// TwinCAT 3 PLC project TcLog
// Title: TcLog
// Company: Benedikt Geisler
// Author: Benedikt Geisler
// ProjectVersion: 0.2.2
// Description: TcLog provides logging functionality to TwinCAT.
// ProgramVersion: 3.1.4023.0
// libraries:
//   Base Interfaces,newest,System
//   Tc2_Standard, * (Beckhoff Automation GmbH)
//   Tc2_System, * (Beckhoff Automation GmbH)
//   Tc2_Utilities, * (Beckhoff Automation GmbH)
//   Tc3_DynamicMemory, * (Beckhoff Automation GmbH)
//   Tc3_Module, * (Beckhoff Automation GmbH)
// project tree:
//   / CONSTANTS.TcGVL
//   Helper functions/ ANY_TO_STRING2.TcPOU, DeleteOldFiles.TcPOU, DynamicStringBuffer.TcPOU, GenerateTimeData.TcPOU, GetFileAgeInSeconds.TcPOU
//   Helper functions/_DataTypes/ DeleteFilesState.TcDUT, PersistToFileState.TcDUT (not stored)
//   Logger/DUT/ E_ErrorCode.TcDUT, E_LogLevel.TcDUT, E_RollingInterval.TcDUT, ST_Error.TcDUT, ST_LoggingConfiguration.TcDUT
//   Logger/ITF/ ILog.TcIO, ILogCore.TcIO
//   Logger/POU/ LogLevel_To_AdsLogMsgType.TcPOU, TcLog.TcPOU, TcLogCore.TcPOU, TcLogTRIG.TcPOU
//   StringBuilder/ ILimitedStringBuilder.TcIO, IStringBuilder.TcIO, StringBuilder.TcPOU
//   Version/ Global_Version.TcGVL
// (motion and I/O tree: see PLC project tclogtest)
// real-time tasks:
//   TASK PlcTask: cycle T#10ms, priority 20, ADS port 350

// ---- Helper functions/_DataTypes/DeleteFilesState.TcDUT
{attribute 'qualified_only'}
{attribute 'strict'}
TYPE INTERNAL DeleteFilesState :
(
	Idle := 0,
  SearchNextFile,
  WaitUntilExecutionDone,
  ProcessFoundFiles,
  CheckIfFileIsDirectory,
  CheckFileTime,
  DeleteFile,
  FileDeleted
);
END_TYPE

// ---- Logger/DUT/E_ErrorCode.TcDUT
{attribute 'qualified_only'}
{attribute 'strict'}
{attribute 'to_string'}
// Provides error return codes for TcLogCore
TYPE E_ErrorCode : 
(
	None,
	OpeningFileFailed,
	WritingToFileFailed,
	ClosingFileFailed,
	EnumeratingFilesInSpecifiedDirectoryFailed,
	DeletingFileFailed,
	FifoOverflow
);
END_TYPE

// ---- Logger/DUT/E_LogLevel.TcDUT
{attribute 'qualified_only'}
{attribute 'strict'}
{attribute 'to_string'}
// Log level of message to be logged.
TYPE E_LogLevel :
(
	Debug,
	Information,
	Warning,
	Error,
	Fatal
);
END_TYPE

// ---- Logger/DUT/E_RollingInterval.TcDUT
{attribute 'qualified_only'}
{attribute 'strict'}
{attrivute 'to_string'}
// Rolling interval to create a new log file when expired. 
TYPE E_RollingInterval :
(
	None,
	Hourly,
	Daily,
	Monthly
);
END_TYPE

// ---- Logger/DUT/ST_Error.TcDUT
TYPE ST_Error :
STRUCT
	Active : BOOL; // TRUE = error is active
	Code : INT; // Error return code => E_ErrorCode
	Info : Tc2_System.T_MaxString; // Error message
END_STRUCT
END_TYPE

// ---- Logger/DUT/ST_LoggingConfiguration.TcDUT
// Configuration of TcLog
TYPE ST_LoggingConfiguration :
STRUCT
	FileName : STRING;
	FilePath : Tc2_System.T_MaxString;
	IncludeInstancePath : BOOL;
	WriteToAds : BOOL;
	RollingInterval : E_RollingInterval;
	MinimumLevel : E_LogLevel;
	Delimiter : STRING(1);
	LogFileLifespan : UINT;
	TimestampFormat : STRING;
END_STRUCT
END_TYPE

// ---- CONSTANTS.TcGVL
{attribute 'qualified_only'}
VAR_GLOBAL CONSTANT
	BUFFER_SIZE : INT := (100 * UDINT_TO_INT(MAX_STRING_LENGTH));
END_VAR

// ---- Version/Global_Version.TcGVL
{attribute 'TcGenerated'}
{attribute 'no-analysis'}
{attribute 'linkalways'}
// This function has been automatically generated from the project information.
VAR_GLOBAL CONSTANT
	{attribute 'const_non_replaced'}
	stLibVersion_TcLog : ST_LibVersion := (iMajor := 0, iMinor := 2, iBuild := 2, iRevision := 0, nFlags := 1, sVersion := '0.2.2');
END_VAR

// ---- Logger/ITF/ILog.TcIO
INTERFACE ILog

METHOD SetLogger : BOOL
VAR_INPUT
	Ref2Core : ILogCore;
END_VAR
END_METHOD

END_INTERFACE

// ---- Logger/ITF/ILogCore.TcIO
INTERFACE ILogCore

// Logger method.
// Logs data in custom format. No additional formatting will be done.
METHOD LogCustomFormat : BOOL
VAR_INPUT
	Data : Tc2_System.T_MaxString; // Data to be logged. No additional formatting will be done.
END_VAR
END_METHOD

// Logger method.
// Logs in the standard format. This includes
// - timestamp
// - log level
// - log message
// - instance path of logging source (optional)
// The message will only be logged if the logging level exceeds the configured minimum logging level.
METHOD LogStandardFormat : BOOL
VAR_INPUT
	Data : Tc2_System.T_MaxString; // Data to be logged. Additional formatting wil be done.
	InstancePath : Tc2_System.T_MaxString; // Instance path of calling logger to locate source of logging message.
	LogLevel : E_LogLevel; // Log level of message.
END_VAR
END_METHOD

END_INTERFACE

// ---- StringBuilder/ILimitedStringBuilder.TcIO
INTERFACE INTERNAL ILimitedStringBuilder

METHOD Append : IStringBuilder // Append text TO t current build STRING.
VAR_INPUT
    Text : Tc2_System.T_MaxString; //Text to append to current build string
END_VAR
END_METHOD

METHOD AppendIf : IStringBuilder
VAR_INPUT
    Condition : BOOL;
    Text : Tc2_System.T_MaxString;
END_VAR
END_METHOD

METHOD Reset : ILimitedStringBuilder //Reset current build STRING TO an empty STRING.
END_METHOD

METHOD ToString : Tc2_System.T_MaxString //Returns current build STRING.
END_METHOD

END_INTERFACE

// ---- StringBuilder/IStringBuilder.TcIO
INTERFACE IStringBuilder

METHOD  Append : IStringBuilder // Append text to t current build string.
VAR_INPUT
	text : Tc2_System.T_MaxString; //Text to append to current build string
END_VAR
END_METHOD

METHOD AppendIf : IStringBuilder
VAR_INPUT
	condition	:	BOOL;
	text : Tc2_System.T_MaxString;
END_VAR
END_METHOD

METHOD InsertAtLocation : IStringBuilder
VAR_INPUT
	Text : Tc2_System.T_MaxString;
	Position:INT;
END_VAR
END_METHOD

METHOD PadLeft : IStringBuilder
VAR_INPUT
	text : Tc2_System.T_MaxString; // Text to append to current build string
	length : INT; // Total length of text + padding
	char : STRING(1); // Character to be padded left of text
END_VAR
END_METHOD

METHOD Reset : ILimitedStringBuilder //Reset current build string to an empty string.
END_METHOD

METHOD ToString : Tc2_System.T_MaxString //Returns current build string.
END_METHOD

END_INTERFACE

// ---- Helper functions/ANY_TO_STRING2.TcPOU
// Converts value of ANY to String.
FUNCTION ANY_TO_STRING2 : T_MAXSTRING
VAR_INPUT
	Data:	ANY;
END_VAR
VAR
	pAnyReal : POINTER TO REAL;
	pAnyLReal: POINTER TO LREAL;	
	pAnyDateAndTime : POINTER TO DATE_AND_TIME;
	pAnyDate: POINTER TO DATE;
	pAnyTime: POINTER TO TIME;
	pAnyWString: POINTER TO WSTRING;
	pAnyTOD: POINTER TO TOD;
	pAnyString: POINTER TO STRING;
	sString: T_MAXSTRING;
	wWString: WSTRING;
END_VAR

IF Data.TypeClass = __SYSTEM.TYPE_CLASS.TYPE_REAL THEN
	pAnyReal := Data.pValue;
	ANY_TO_STRING2 := REAL_TO_STRING(pAnyReal^);
	
ELSIF Data.TypeClass = __SYSTEM.TYPE_CLASS.TYPE_LREAL THEN
	pAnyLReal := Data.pValue;
	ANY_TO_STRING2 := LREAL_TO_STRING(pAnyLReal^);
	
ELSIF Data.TypeClass = __SYSTEM.TYPE_CLASS.TYPE_DATEANDTIME THEN
	pAnyDateAndTime := Data.pValue;
	ANY_TO_STRING2 := DT_TO_STRING(pAnyDateAndTime^);	
	
ELSIF Data.TypeClass = __SYSTEM.TYPE_CLASS.TYPE_DATE THEN
	pAnyDate := Data.pValue;
	ANY_TO_STRING2 := DATE_TO_STRING(pAnyDate^);
	
ELSIF Data.TypeClass = __SYSTEM.TYPE_CLASS.TYPE_TIME THEN
	pAnyTime := Data.pValue;
	ANY_TO_STRING2 := TIME_TO_STRING(pAnyTime^);
	
ELSIF Data.TypeClass = __SYSTEM.TYPE_CLASS.TYPE_STRING THEN
	pAnyString := Data.pValue;
	ANY_TO_STRING2 := pAnyString^;
	
ELSIF Data.TypeClass = __SYSTEM.TYPE_CLASS.TYPE_WSTRING THEN
	pAnyWString := Data.pValue;
	wWString := pAnyWString^;
	WSTRING_TO_STRING2(ADR(sString), ADR(wWstring), SIZEOF(wWString));
	ANY_TO_STRING2 := sString;
	
ELSIF Data.TypeClass = __SYSTEM.TYPE_CLASS.TYPE_TIMEOFDAY THEN
	pAnyTOD := Data.pValue;
	ANY_TO_STRING2 := TOD_TO_STRING(pAnyTOD^);
	
ELSE
	ANY_TO_STRING2 := ANY_TO_STRING(Data.pValue^);
END_IF

END_FUNCTION

// ---- Helper functions/DeleteOldFiles.TcPOU
FUNCTION_BLOCK DeleteOldFiles
VAR_INPUT
	StartScan : BOOL; // Rising edge starts scan for out-of-date log files and deletes them.
	ExpirationInDays : UINT; // Files will be deleted if older than n days
	FilePath : Tc2_System.T_MaxString; // Path to files to be deleted
	FileName : Tc2_System.T_MaxString; // Only files which match this filename will be deleted
	ActualTime : Tc2_Utilities.T_FILETIME; // Actual Time 
END_VAR
VAR_OUTPUT
	Error : ST_Error; // Error information
END_VAR
VAR CONSTANT
	ONE_DAY_IN_SECONDS : LREAL := 24*3600.0;
	MAX_NUMBER_OF_FILES : UDINT := 100;
END_VAR
VAR
	state : DeleteFilesState := DeleteFilesState.Idle;
  
	fbEnum : Tc2_Utilities.FB_EnumFindFileList;
	fTrigEnumBusy : Tc2_Standard.F_TRIG;
	fbDeleteFile : Tc2_System.FB_FileDelete;
	fTrigDeleteFileBusy : Tc2_Standard.F_TRIG;
	filesList : ARRAY[1..100] OF Tc2_Utilities.ST_FindFileEntry;
	deleteFileIndex : UDINT;
	deleteFileName : Tc2_System.T_MaxString;
	eEnumCmd : Tc2_Utilities.E_EnumCmdType;
	bFileDeleted : BOOL;
END_VAR
VAR_TEMP
	timeLastWriteAccess : Tc2_Utilities.T_ULARGE_INTEGER;
	fileTimeAsULINT : Tc2_Utilities.T_ULARGE_INTEGER;
	fileTimeDifference : Tc2_Utilities.T_ULARGE_INTEGER;
END_VAR

// State machine to delete all due files.
// It first enumerates all files in the specified directory
// and then deletes all files that have overpassed the specified due date
CASE state OF
	DeleteFilesState.Idle:
		IF StartScan THEN
			eEnumCmd:= eEnumCmd_First;
			deleteFileIndex := 1;
			state := DeleteFilesState.SearchNextFile;
		END_IF
		
	DeleteFilesState.SearchNextFile:
		IF fTrigEnumBusy.Q THEN
			state := DeleteFilesState.WaitUntilExecutionDone;
		END_IF
		
	DeleteFilesState.WaitUntilExecutionDone:
		IF NOT fbEnum.bError THEN
			IF NOT fbEnum.bEOE THEN
				IF fbEnum.nFindFiles < MAX_NUMBER_OF_FILES THEN
					State := DeleteFilesState.SearchNextFile;
				ELSE
					eEnumCmd := eEnumCmd_Abort;
					state := DeleteFilesState.ProcessFoundFiles;
				END_IF
			ELSE
				state := DeleteFilesState.ProcessFoundFiles;
			END_IF
		ELSE
			state := DeleteFilesState.Idle;
		END_IF
		
	DeleteFilesState.ProcessFoundFiles:
		IF deleteFileIndex > fbEnum.nFindFiles THEN
			state := DeleteFilesState.Idle;
		ELSE
			state := DeleteFilesState.CheckIfFileIsDirectory;
		END_IF
		
	DeleteFilesState.CheckIfFileIsDirectory:
		IF NOT filesList[deleteFileIndex].fileAttributes.bDirectory THEN
			state := DeleteFilesState.CheckFileTime;
		ELSE
			deleteFileIndex := deleteFileIndex + 1;
			state := DeleteFilesState.ProcessFoundFiles;
		END_IF
		
	DeleteFilesState.CheckFileTime:		
		IF GetFileAgeInSeconds(ActualTime, filesList[deleteFileIndex]) > (ExpirationInDays * ONE_DAY_IN_SECONDS) THEN
			state := DeleteFilesState.DeleteFile;
		ELSE
			deleteFileIndex := deleteFileIndex + 1;
			state := DeleteFilesState.ProcessFoundFiles;
		END_IF
	
	DeleteFilesState.DeleteFile:
		deleteFileName := CONCAT(FilePath, filesList[deleteFileIndex].sFileName);
		
		IF fTrigDeleteFileBusy.Q THEN
			deleteFileIndex := deleteFileIndex + 1;
			bFileDeleted := TRUE;
			state := DeleteFilesState.FileDeleted;
		END_IF
		IF fbDeleteFile.bError THEN
			state := DeleteFilesState.Idle;
		END_IF
		
	DeleteFilesState.FileDeleted:		
		// This state is needed to generate a rising edge for FB_FileDelete
		IF NOT bFileDeleted THEN
			state := DeleteFilesState.ProcessFoundFiles;
		END_IF
		bFileDeleted := FALSE;

END_CASE

// Function blocks used in state machine

// Search files in given directory
fbEnum(sNetId := '',
       eCmd := eEnumCmd,
       sPathName := CONCAT(FilePath, CONCAT('*', FileName)),
       bExecute := (state = DeleteFilesState.SearchNextFile) OR (eEnumCmd = eEnumCmd_Abort AND state <> DeleteFilesState.Idle),
       pFindList := ADR(filesList),
       cbFindList := SIZEOF(filesList),
       tTimeout := T#10S);

fTrigEnumBusy(CLK:=fbEnum.bBusy);

// Delete files
fbDeleteFile(sNetId := '',
             sPathName := deleteFileName,
             bExecute := (state = DeleteFilesState.DeleteFile),
             tTimeout := T#10S);
				
fTrigDeleteFileBusy(CLK := fbDeleteFile.bBusy);

// Error handling
Error.Active := FALSE;
Error.Code := E_ErrorCode.None;
Error.Info := '';

IF fbEnum.bError THEN
	Error.Active := TRUE;
	Error.Code := E_ErrorCode.EnumeratingFilesInSpecifiedDirectoryFailed;
	Error.Info := CONCAT('Enumerating files in specified directory failed. Error thrown by FB_EnumFindFileList. Consult Beckhoff InfoSys. Internal Error: ', UDINT_TO_STRING(fbEnum.nErrId));
END_IF
			
IF fbDeleteFile.bError THEN
	Error.Active := TRUE;
	Error.Code := E_ErrorCode.DeletingFileFailed;
	Error.Info := CONCAT('Deleting expired log file in specified directory failed. Error thrown by FB_FileDelete. Consult Beckhoff InfoSys. Internal Error: ', UDINT_TO_STRING(fbDeleteFile.nErrId));
END_IF

END_FUNCTION_BLOCK

// ---- Helper functions/GetFileAgeInSeconds.TcPOU
FUNCTION GetFileAgeInSeconds : DINT
VAR_INPUT
	ActualTime : Tc2_Utilities.T_FILETIME;
	FindFileEntry	: Tc2_Utilities.ST_FindFileEntry;
END_VAR
VAR
	timeLastWriteAccess : Tc2_Utilities.T_ULARGE_INTEGER;
	fileTimeAsULINT : Tc2_Utilities.T_ULARGE_INTEGER;
	fileTimeDifference : Tc2_Utilities.T_ULARGE_INTEGER;
END_VAR

// Local file time
fileTimeAsULINT.dwLowPart := ActualTime.dwLowDateTime;
fileTimeAsULINT.dwHighPart := ActualTime.dwHighDateTime;

// Write access is UTC
timeLastWriteAccess.dwLowPart := FindFileEntry.lastWriteTime.dwLowDateTime;
timeLastWriteAccess.dwHighPart := FindFileEntry.lastWriteTime.dwHighDateTime;
fileTimeDifference := UInt64Sub64(fileTimeAsULINT, timeLastWriteAccess);

GetFileAgeInSeconds := LREAL_TO_DINT(UINT64_TO_LREAL(fileTimeDifference)/(1000*1000*10));

END_FUNCTION

// ---- Helper functions/DynamicStringBuffer.TcPOU
FUNCTION_BLOCK DynamicStringBuffer
VAR_OUTPUT
	Error : ST_ERROR; // Error information of this FB
END_VAR
VAR
	Fifo : Tc2_Utilities.FB_StringRingBuffer; // Necessary to buffer log data until it has been written to file.
	MemMan : Tc3_DynamicMemory.FB_DynMem_Manager; // Memory manager, required by DynMem_Buffer.
	MemBuf : Tc3_DynamicMemory.FB_DynMem_Buffer(ipMemMan := MemMan); // Provides dynamic buffer for Fifo. Is extended automatically if more than the 
                                                                   // default buffer size is needed.
	{attribute 'hide'} 														
	_busy : BOOL; // Buffer is busy; typically with writing data to the file system.
END_VAR

METHOD AddLine : BOOL
VAR_INPUT
	Text : Tc2_System.T_MaxString; // Text to be added to the buffer
END_VAR
ResizeFifoBufferIfNecessary();
Fifo.A_AddTail(putValue := CONCAT(Text, '$N'));
END_METHOD

METHOD AddString : BOOL
VAR_INPUT
	Text : Tc2_System.T_MaxString; // String to be added to the buffer
END_VAR
ResizeFifoBufferIfNecessary();
Fifo.A_AddTail(putValue := Text);
END_METHOD

METHOD PRIVATE AllocateBuffer : BOOL	// Allocates buffer for the Fifo.
VAR_INPUT
	nbufferSize : UDINT;
END_VAR
MemBuf.CreateBuffer(nSize:=nbufferSize*SIZEOF(BYTE), bReset:=TRUE);
Fifo.pBuffer := MemBuf.pBuffer;
Fifo.cbBuffer := nbufferSize*SIZEOF(BYTE);
END_METHOD

{attribute 'monitoring':='call'}
PROPERTY Busy : BOOL
GET
Busy := _busy;
END_GET
SET // PRIVATE
_busy := Busy;
END_SET
END_PROPERTY

METHOD FB_exit : BOOL
VAR_INPUT
	bInCopyCode : BOOL; // if TRUE, the exit method is called for exiting an instance that is copied afterwards (online change).
END_VAR
MemBuf.Clear();
END_METHOD

METHOD FlushCache : BOOL
Fifo.A_Reset();
END_METHOD

METHOD INTERNAL Init : BOOL
VAR_INPUT
	nBufferSize : UDINT; // Buffer size for the string buffer
END_VAR
AllocateBuffer(nBufferSize);
END_METHOD

METHOD PersistToFile : BOOL
VAR_INPUT
	FileName : Tc2_System.T_MaxString; // File name including its path
END_VAR
VAR_INST
	state : PersistToFileState;		
		
	fbFileOpen : Tc2_System.FB_FileOpen;
	hFile : UINT;
	               	
	fbFileWrite : Tc2_System.FB_FileWrite;
	lockFileWriteToForceRisingEdge : BOOL; // filePuts can only be executed every other cycle
                                         // since it needs a rising edge to execute.
	fbFileClose : Tc2_System.FB_FileClose;
	
	buffer : ARRAY[0..CONSTANTS.BUFFER_SIZE] OF BYTE;
	currentBufferPos : UDINT;
	fifoHeadString : Tc2_System.T_MaxString;
	fifoHeadLength : UDINT;
	fifoHeadBytes : ARRAY[0..MAX_STRING_LENGTH] OF BYTE;
	i : UINT;
END_VAR
VAR CONSTANT
  NET_ID : STRING := '';
	TIMEOUT : TIME := DEFAULT_ADS_TIMEOUT;
	MAX_LOGS_PER_CYCLE : UINT := DINT_TO_UINT(CONSTANTS.BUFFER_SIZE / UDINT_TO_DINT(MAX_STRING_LENGTH));
	MAX_BUFFER_POS : UDINT := (SIZEOF(buffer) - MAX_STRING_LENGTH);
END_VAR
// State machine
// Using if-statements instead of case for performance reasons:
// Some states execute instantly and allow thus the next state 
// to start within the same plc cycle.

// *** I D L E ***
IF state = PersistToFileState.Idle THEN
	lockFileWriteToForceRisingEdge := FALSE;
	IF Fifo.nCount > 0 THEN 
		lockFileWriteToForceRisingEdge := FALSE;
		state := PersistToFileState.OpenFile;
	END_IF
END_IF
		
// *** O P E N   F I L E ***
fbFileOpen(sNetId := NET_ID, sPathName := FileName, nMode := FOPEN_MODEAPPEND OR FOPEN_MODETEXT, 
	         ePath := PATH_GENERIC, bExecute := (state = PersistToFileState.OpenFile), tTimeout := TIMEOUT,
	         hFile => hFile);

IF state = PersistToFileState.OpenFile THEN
	IF fbFileOpen.bError THEN
		state := PersistToFileState.CloseFile;
	ELSIF NOT fbFileOpen.bBusy THEN 
		state := PersistToFileState.GetStringFromFifo; 
	END_IF
END_IF 

// *** P O P   F R O M   F I F O ***
IF state = PersistToFileState.GetStringFromFifo THEN
	IF NOT lockFileWriteToForceRisingEdge THEN
		currentBufferPos := 0;
		FOR i:=0 TO MAX_LOGS_PER_CYCLE DO
			IF Fifo.nCount <= 0 THEN EXIT; END_IF
			IF currentBufferPos >= MAX_BUFFER_POS THEN EXIT; END_IF
			
			Fifo.A_RemoveHead(getValue => fifoHeadString);	
			fifoHeadBytes := MAXSTRING_TO_BYTEARR(fifoHeadString);
			fifoHeadLength := INT_TO_UDINT(LEN(fifoHeadString));
			MEMCPY(
				destAddr 	:= 	ADR(buffer) + SIZEOF(BYTE) * currentBufferPos,
				srcAddr 	:=	ADR(fifoHeadBytes),
				n			:=	fifoHeadLength);		
			currentBufferPos := currentBufferPos + fifoHeadLength; 	
		END_FOR
		state := PersistToFileState.AppendDataToFile;
	END_IF
	lockFileWriteToForceRisingEdge := FALSE;
END_IF
	
// *** W R I T E   T O   F I L E ***
fbFileWrite(
	sNetId := NET_ID, 
	hFile := hFile, 
	pWriteBuff := ADR(buffer),
	cbWriteLen := currentBufferPos,
	bExecute := state = PersistToFileState.AppendDataToFile, 
	tTimeout := TIMEOUT);	

IF state = PersistToFileState.AppendDataToFile THEN
	lockFileWriteToForceRisingEdge := TRUE;		
	IF fbFileWrite.bError THEN
		state := PersistToFileState.CloseFile;
	ELSIF Fifo.nCount > 0 AND NOT fbFileWrite.bBusy THEN
		state := PersistToFileState.GetStringFromFifo; 
	ELSIF Fifo.nCount = 0 THEN
		state := PersistToFileState.CloseFile;
	END_IF
END_IF
		
// *** C L O S E   F I L E ***
fbFileClose(
	sNetId := NET_ID, hFile := hFile, 
	bExecute := (state = PersistToFileState.CloseFile), tTimeout := TIMEOUT);

IF state = PersistToFileState.CloseFile THEN
	IF NOT fbFileCLose.bBusy THEN state := PersistToFileState.Idle; END_IF
END_IF

// Close file in case of error
IF fbFileOpen.bError THEN state := PersistToFileState.CloseFile; END_IF
IF fbFileWrite.bError THEN state := PersistToFileState.CloseFile; END_IF
IF NOT Fifo.bOk AND Fifo.nCount > 0 AND state <> PersistToFileState.Idle THEN 
	state := PersistToFileState.CloseFile; 
END_IF

// Error handling
IF fbFileOpen.bError THEN
	Error.Active := TRUE;
	Error.Code := E_ErrorCode.OpeningFileFailed;
	Error.Info := CONCAT('Opening file failed. Error thrown by FB_FileOpen. Consult Beckhoff InfoSys. Internal Error: ', UDINT_TO_STRING(fbFileOpen.nErrId));
ELSIF fbFileWrite.bError THEN
	Error.Active := TRUE;
	Error.Code := E_ErrorCode.WritingToFileFailed;
	Error.Info := CONCAT('Writing to file failed. Error thrown by FB_FileWrite. Consult Beckhoff InfoSys. Internal Error: ', UDINT_TO_STRING(fbFileWrite.nErrId));
ELSIF fbFileClose.bError THEN
	Error.Active := TRUE;
	Error.Code := E_ErrorCode.ClosingFileFailed;
	Error.Info := CONCAT('Closing file failed. Error thrown by FB_FileClose. Consult Beckhoff InfoSys. Internal Error: ', UDINT_TO_STRING(fbFileClose.nErrId));
ELSIF NOT Fifo.bOk AND Fifo.nCount > 0 THEN
	Error.Active := TRUE;
	Error.Code := E_ErrorCode.FifoOverflow;
	Error.Info := 'FIFO overflow. Check if plc has enough free memory.';
ELSE
	Error.Active := FALSE;
	Error.Code := E_ErrorCode.None;
	Error.Info := '';
END_IF

// Set busy state
Busy := (state <> PersistToFileState.Idle OR Fifo.nCount > 0);

(* Uncomment for cyclic logging of state machine, buffer usage & errors

ADSLOGSTR(ADSLOG_MSGTYPE_LOG, 
	CONCAT('****DynamicStringBuffer.state:', 
	CONCAT(UINT_TO_STRING(state),
	CONCAT(', DynamicStringBuffer.hFile:', UINT_TO_STRING(hFile)))), '');

ADSLOGSTR(ADSLOG_MSGTYPE_LOG, 
	CONCAT('****Fifo: used ', 
	CONCAT(UDINT_TO_STRING(Fifo.cbSize),
	CONCAT(' of ', UDINT_TO_STRING(Fifo.cbBuffer)))), '');
	
IF Error.Active THEN
	ADSLOGSTR(ADSLOG_MSGTYPE_LOG, 
		CONCAT('****DynamicStringBuffer.Error: ', Error.Info), 
		'');	
END_IF
*)
END_METHOD

METHOD PopHead : Tc2_System.T_MaxString
VAR_INST
	headString : Tc2_System.T_MaxString;
END_VAR
Fifo.A_RemoveHead(getValue => headString);
PopHead := headString;
END_METHOD

// Resizes the buffer for the FIFO if necessary
METHOD PRIVATE ResizeFifoBufferIfNecessary : BOOL
VAR
	requiredSize : UDINT;
	newSize : DINT;
END_VAR
requiredSize := Fifo.cbSize + MAX_STRING_LENGTH;

IF requiredSize > Fifo.cbBuffer THEN
	MemBuf.Resize(nSize := requiredSize*SIZEOF(BYTE), bPreserve:=TRUE, bReset:=TRUE);
	Fifo.pBuffer := MemBuf.pBuffer;
	Fifo.cbBuffer := requiredSize;
END_IF
END_METHOD

END_FUNCTION_BLOCK

// ---- Helper functions/GenerateTimeData.TcPOU
FUNCTION_BLOCK GenerateTimeData
VAR_OUTPUT
	timeAsFileTime : Tc2_Utilities.T_FILETIME;
	timeAsSystemTime : Tc2_Utilities.TIMESTRUCT;
	timeAsString : Tc2_System.T_MaxString;
	utcTimeAsFileTime : Tc2_Utilities.T_FILETIME;
END_VAR
VAR
	fbSystemTime : Tc2_Utilities.FB_LocalSystemTime;
	fbSystemTime1 : Tc2_System.GETSYSTEMTIME;
	fbTimeZoneInfo : Tc2_Utilities.FB_GetTimeZoneInformation;
	fbLocalTime : Tc2_Utilities.FB_SystemTimeToTzSpecificLocalTime;
	rTrigTimeValid : Tc2_Standard.R_TRIG;
	fbUTCTime : Tc2_Utilities.FB_TzSpecificLocalTimeToFileTime;
END_VAR
VAR_TEMP
	utcSystemTime : Tc2_Utilities.TIMESTRUCT;
END_VAR

fbSystemTime(
	sNetID	:=	'',
	bEnable := 	TRUE,
	dwCycle	:=	1,
	dwOpt	:=	1,
	tTimeout:=	DEFAULT_ADS_TIMEOUT
);

fbTimeZoneInfo(
	sNetID := '',
	bExecute := TRUE,
	tTimeout := DEFAULT_ADS_TIMEOUT);

fbUTCTime(
	in := SYSTEMTIME_TO_FILETIME(timeAsSystemTime),
	tzInfo := fbTimeZoneInfo.tzInfo);
	
timeAsSystemTime 	:=	fbSystemTime.systemTime;
timeAsFileTime 		:= 	SYSTEMTIME_TO_FILETIME(timeAsSystemTime);
timeAsString 		:= 	SYSTEMTIME_TO_STRING(timeAsSystemTime);
utcTimeAsFileTime	:= 	fbUTCTime.out;

rTrigTimeValid(CLK := fbSystemTime.bValid);

{attribute 'monitoring':='call'}
PROPERTY Done : BOOL
GET
Done := rTrigTimeValid.Q;
END_GET
END_PROPERTY

// Replaces placeholders in format string by the actual time values
METHOD PRIVATE ReplaceFormatPlaceholder : STRING
VAR_INPUT
	Format : STRING;
	Length : INT;
	TimeType : STRING(1);
END_VAR
VAR_INST
	i : INT;
	replaceString : STRING;
	timeString : STRING;
END_VAR
IF    TimeType = 'Y' 	THEN timeString := TO_STRING(timeAsSystemTime.wYear); 
ELSIF TimeType = 'M' 	THEN timeString := TO_STRING(timeAsSystemTime.wMonth); 
ELSIF TimeType = 'D' 	THEN timeString := TO_STRING(timeAsSystemTime.wDay); 
ELSIF TimeType = 'h' 	THEN timeString := TO_STRING(timeAsSystemTime.wHour); 
ELSIF TimeType = 'm' 	THEN timeString := TO_STRING(timeAsSystemTime.wMinute); 
ELSIF TimeType = 's' 	THEN timeString := TO_STRING(timeAsSystemTime.wSecond); 
ELSIF TimeType = 'i' 	THEN timeString := TO_STRING(timeAsSystemTime.wMilliseconds); 
ELSE
  timeString:='';
END_IF

replaceString := '';

IF Length > LEN(timeString) THEN
	FOR i:=1 TO Length - LEN(timeString) DO
		replaceString := CONCAT(replaceString, '0');
	END_FOR
	replaceString := CONCAT(replaceString, timeString);
ELSE
	replaceString := RIGHT(timeString, Length);
END_IF

ReplaceFormatPlaceholder := REPLACE(Format, replaceString, Length, FIND(Format, TimeType));
END_METHOD

// Returns a formatted string containing the actual time information 
//	Y : year
//	M : month
// 	D : day
//  h : hour 
//  m : minute
//  s : second
//  i : millisecond
// 
// Example: _YYMMDD-hh:mm:ss:iii_
// => _20210812-12:30:22:123_
METHOD ToString : Tc2_System.T_MaxString
VAR_INPUT
	Format : STRING;
END_VAR
VAR_INST
	inputString : STRING;
	char : STRING(1);
  formattedString : Tc2_System.T_MaxString;  
END_VAR
VAR
	year : INT := 0;
	month : INT := 0;
	day : INT := 0;
	hour : INT := 0;
	minute : INT := 0;
	second : INT := 0;
	millisecond : INT := 0;
END_VAR
VAR CONSTANT
	VALID_FORMAT : STRING := 'YMDhms';
END_VAR
// Parses "Format" and returns a adequatly formatted string containing the time information
inputString := Format;

WHILE LEN(inputString) > 0 DO
	char := LEFT(inputString, 1);
	
	IF    char = 'Y' THEN 	year := year + 1;
	ELSIF char = 'M' THEN	month := month + 1;
	ELSIF char = 'D' THEN	day := day + 1;
	ELSIF char = 'h' THEN	hour := hour + 1;
	ELSIF char = 'm' THEN	minute := minute + 1;
	ELSIF char = 's' THEN 	second := second + 1;
	ELSIF char = 'i' THEN 	millisecond := millisecond + 1;
	END_IF
	
	inputString := DELETE(inputString, 1, 1);
END_WHILE

formattedString := ReplaceFormatPlaceholder(Format, year, 'Y');
formattedString := ReplaceFormatPlaceholder(formattedString, month, 'M');
formattedString := ReplaceFormatPlaceholder(formattedString, day, 'D');
formattedString := ReplaceFormatPlaceholder(formattedString, hour, 'h');
formattedString := ReplaceFormatPlaceholder(formattedString, minute, 'm');
formattedString := ReplaceFormatPlaceholder(formattedString, second, 's');
formattedString := ReplaceFormatPlaceholder(formattedString, millisecond, 'i');

ToString := formattedString;
END_METHOD

END_FUNCTION_BLOCK

// ---- Logger/POU/LogLevel_To_AdsLogMsgType.TcPOU
FUNCTION INTERNAL LogLevel_To_AdsLogMsgType : DWORD
VAR_INPUT
	LogLevel : E_LogLevel;
END_VAR
VAR
	retVal : DWORD; 
END_VAR

CASE LogLevel OF
	E_LogLevel.Debug, E_LogLevel.Information:
		retVal := Tc2_System.ADSLOG_MSGTYPE_HINT;
	E_LogLevel.Warning:
		retVal := Tc2_System.ADSLOG_MSGTYPE_WARN;
	E_LogLevel.Error, E_LogLevel.Fatal:
		retVal := Tc2_System.ADSLOG_MSGTYPE_ERROR;
	ELSE
		retVal := Tc2_System.ADSLOG_MSGTYPE_HINT;
END_CASE

LogLevel_To_AdsLogMsgType := retVal;

END_FUNCTION

// ---- Logger/POU/TcLog.TcPOU
{attribute 'reflection'} 
FUNCTION_BLOCK TcLog IMPLEMENTS ILog
VAR
	{attribute 'hide'} 
	logConditionSatisfied : BOOL; // flag that indicates, whether log condition has been satisfied. 
                                // Logging will only be carried out it this evaluates to TRUE.
	{attribute 'hide'} 																
	logDataInitialized : BOOL; // flag that indicate, whether log data has been initialized. 
                             // Necessary for configuration methods to provide a fluent interface.
	{attribute 'hide'} 																
	logData : Tc2_System.T_MaxString; // contains message to be logged.
	
	{attribute 'hide'} 
	usedLogger : ILogCore; // 
	
	{attribute 'instance-path'} 
  {attribute 'noinit'} 
  InstancePath : STRING; // contains instance path 
END_VAR
VAR_STAT
	SingletonInstance : ILogCore; // Wires up TcLog ("Client") to TcLogCore ("Server") (Singleton-Behaviour)
END_VAR

// Appends any given data to the log string. Can be chained.
METHOD AppendAny : REFERENCE TO TcLog	
VAR_INPUT
	Data : ANY; // Data to be appended to log string.
END_VAR
VAR
	pAnyReal : POINTER TO REAL;
	pAnyLReal : POINTER TO LREAL;
END_VAR
InitializeLogData();

logData := CONCAT(logData, ANY_TO_STRING2(Data));

AppendAny REF= THIS^;
END_METHOD

// Appends a string to the log string. Can be chained.
METHOD AppendString : REFERENCE TO TcLog		
VAR_INPUT
	Data : Tc2_System.T_MaxString; // Data to be appended to log string.
END_VAR
InitializeLogData();

logData := Tc2_Standard.CONCAT(logData, Data);
	
AppendString REF= THIS^;
END_METHOD

// Appends information about the given variable to the log string. 
// Can be chained.
// Example: 
// ---------------
// VAR
// 		myInt : INT := 10;
//		myVarInfo : __SYSTEM.VAR_INFO := __VARINFO(myInt);
// END_VAR
// Logger.AppendVariable(myVarInfo, myInt);
METHOD AppendVariable : REFERENCE TO TcLog		
VAR_INPUT
	VarInfo : 	__SYSTEM.VAR_INFO; // VARINFO of variable to be appended to log string.
	Value : ANY; // Value of variable to be appended to log string.
END_VAR
VAR
	Format : Tc2_Utilities.FB_FormatString;
	symbolName : Tc2_System.T_MaxString;
	typeName : Tc2_System.T_MaxString; 
END_VAR
InitializeLogData();

symbolName := VarInfo.Symbol;
typeName := VarInfo.TypeName; 

Format(
	sFormat := '%s [%s] : ',
	arg1 := Tc2_Utilities.F_STRING(symbolName),
	arg2 := Tc2_Utilities.F_STRING(typeName));
	
AppendString(Format.sOut);
AppendAny(Value);

AppendVariable REF= THIS^;
END_METHOD

//	Logs the log string in DEBUG level
METHOD Debug : BOOL	
VAR_INPUT
	Message	:	Tc2_System.T_MaxString; // Message to be appended to log string.
END_VAR
InitializeLogData();
IF logConditionSatisfied THEN
	IF usedLogger <> 0 THEN 
		usedLogger.LogStandardFormat(CONCAT(logData, Message), ShortenInstancePath(InstancePath), E_LogLevel.Debug); 
	ELSE
		ADSLOGSTR(ADSLOG_MSGTYPE_LOG OR LogLevel_To_AdsLogMsgType(E_LogLevel.Error), 'usedLogger: No valid reference', ''); 
	END_IF
END_IF
logDataInitialized := FALSE;
END_METHOD

// Logs the log string in ERROR level
METHOD Error : BOOL	
VAR_INPUT
	Message	:	Tc2_System.T_MaxString; // Message to be appended to log string.
END_VAR
InitializeLogData();
IF logConditionSatisfied THEN
	IF usedLogger <> 0 THEN 
		usedLogger.LogStandardFormat(CONCAT(logData, Message), ShortenInstancePath(InstancePath), E_LogLevel.Error); 
	ELSE
		ADSLOGSTR(ADSLOG_MSGTYPE_LOG OR LogLevel_To_AdsLogMsgType(E_LogLevel.Error), 'usedLogger: No valid reference', ''); 
	END_IF
END_IF
logDataInitialized := FALSE;
END_METHOD

// Logs the log string in FATAL level
METHOD Fatal : BOOL		
VAR_INPUT
	Message	:	Tc2_System.T_MaxString; // Message to be appended to log string.
END_VAR
InitializeLogData();
IF logConditionSatisfied THEN
	IF usedLogger <> 0 THEN 
		usedLogger.LogStandardFormat(CONCAT(logData, Message), ShortenInstancePath(InstancePath), E_LogLevel.Fatal); 
	ELSE
		ADSLOGSTR(ADSLOG_MSGTYPE_LOG OR LogLevel_To_AdsLogMsgType(E_LogLevel.Error), 'usedLogger: No valid reference', ''); 
	END_IF
END_IF
logDataInitialized := FALSE;
END_METHOD

// Logs the log string in INFORMATION level.
METHOD Information : BOOL
VAR_INPUT
	Message	:	Tc2_System.T_MaxString; // Message to be appended to log string.
END_VAR
InitializeLogData();
IF logConditionSatisfied THEN
	IF usedLogger <> 0 THEN 
		usedLogger.LogStandardFormat(CONCAT(logData, Message), ShortenInstancePath(InstancePath), E_LogLevel.Information); 
	ELSE
		ADSLOGSTR(ADSLOG_MSGTYPE_LOG OR LogLevel_To_AdsLogMsgType(E_LogLevel.Error), 'usedLogger: No valid reference', ''); 
	END_IF
END_IF
logDataInitialized := FALSE;
END_METHOD

// Initializes the reference to the core logger. Should only be called once from the core logger directly.
METHOD PUBLIC Init : BOOL		
VAR_INPUT
	Ref2Core : ILogCore; // Reference to TcLoggerCore instance.
END_VAR
SingletonInstance := Ref2Core;
END_METHOD

// Necessary to provide a fluent interface of the function. 
// Has to be called at the begin of any method that returns a reference to THIS^
{attribute 'hide'}
METHOD PRIVATE InitializeLogData : BOOL
IF NOT logDataInitialized THEN
	logConditionSatisfied := TRUE;
	logData := '';
	logDataInitialized := TRUE;
	IF usedLogger = 0 THEN usedLogger := SingletonInstance; END_IF
END_IF
END_METHOD

// Conditional execution of the log commant. Only executes logging when Cond = TRUE.
METHOD OnCondition : REFERENCE TO TcLog
VAR_INPUT
	Cond: BOOL; // Logs data only if this condition evaluates to TRUE.
END_VAR
InitializeLogData();

logConditionSatisfied := Cond;

OnCondition REF= THIS^;
END_METHOD

// Initializes the reference to the core logger. Should only be called once from the core logger directly.
METHOD SetLogger : BOOL
VAR_INPUT
	Ref2Core : ILogCore; // Reference to Core Logger
END_VAR
usedLogger := Ref2Core;
END_METHOD

// Helper method. Shortens the instance path by omitting superfluent information
// such as concrete logger instance and plc/project names.
{attribute 'hide'}
METHOD PRIVATE ShortenInstancePath : Tc2_System.T_MaxString
VAR_INPUT
	Path : Tc2_System.T_MaxString; // Instance path to be shortened.
END_VAR
VAR
	i : UINT;
	shortenedPath : Tc2_System.T_MaxString;
	positionInString : INT := 0;
	positionOfLastDot : INT := 0;
END_VAR
shortenedPath := Path;

// Find last '.'
WHILE(FIND(shortenedPath, '.') > 0) DO
	positionInString := FIND(shortenedPath, '.');
	shortenedPath := DELETE(shortenedPath, positionInString+1, 0);	
	positionOfLastDot := positionOfLastDot+positionInString;
END_WHILE

shortenedPath := Path;
// Delete instantiation of this FB (obvious information)
shortenedPath := DELETE(shortenedPath, LEN(shortenedPath)-positionOfLastDot+1, positionOfLastDot);
// Delete project information
positionInString := FIND(shortenedPath, '.');
shortenedPath := DELETE(shortenedPath, positionInString+1, 0);
// Delete PLC information
positionInString := FIND(shortenedPath, '.');
shortenedPath := DELETE(shortenedPath, positionInString+1, 0);

ShortenInstancePath := shortenedPath;
END_METHOD

// Logs directly to ADS log, ignoring the settings of the base logger.
METHOD ToAdsLog : BOOL
VAR_INPUT
	LogLevel : E_LogLevel; // Log level in which message should be logged to ADS.
END_VAR
InitializeLogData();

IF logConditionSatisfied THEN
	ADSLOGSTR(ADSLOG_MSGTYPE_LOG OR LogLevel_To_AdsLogMsgType(LogLevel), logData, ''); 
END_IF

logDataInitialized := FALSE;
END_METHOD

// Saves custom formatted log string. No addtitional information will be added.
METHOD ToCustomFormat : BOOL
VAR_INPUT
	Message	:	Tc2_System.T_MaxString; // Message to be appended to log string.
END_VAR
InitializeLogData();
IF logConditionSatisfied THEN
	IF usedLogger <> 0 THEN 
		usedLogger.LogCustomFormat(CONCAT(logData, Message)); 
	ELSE
		ADSLOGSTR(ADSLOG_MSGTYPE_LOG OR LogLevel_To_AdsLogMsgType(E_LogLevel.Error), 'usedLogger: No valid reference', ''); 
	END_IF
END_IF
logDataInitialized := FALSE;
END_METHOD

// Logs the log string in WARNING level
METHOD Warning : BOOL	
VAR_INPUT
	Message	:	Tc2_System.T_MaxString; // Message to be appended to log string.
END_VAR
InitializeLogData();
IF logConditionSatisfied THEN
	IF usedLogger <> 0 THEN 
		usedLogger.LogStandardFormat(CONCAT(logData, Message), ShortenInstancePath(InstancePath), E_LogLevel.Warning); 
	ELSE
		ADSLOGSTR(ADSLOG_MSGTYPE_LOG OR LogLevel_To_AdsLogMsgType(E_LogLevel.Error), 'usedLogger: No valid reference', ''); 
	END_IF
END_IF
logDataInitialized := FALSE;
END_METHOD

END_FUNCTION_BLOCK

// ---- Logger/POU/TcLogCore.TcPOU
FUNCTION_BLOCK TcLogCore IMPLEMENTS ILogCore
VAR
	{attribute 'hide'} 
	LoggingSingleton : TcLog;	// Logger-Singleton: Required to provide Singleton-functionality for TcLog.
	{attribute 'hide'} 			
	timeAsFileTime : Tc2_Utilities.T_FILETIME; // Actual time as filetime, corrected to local time zone
	{attribute 'hide'} 			
	utcTimeAsFileTime : Tc2_Utilities.T_FILETIME; // Actual time as filetime
	{attribute 'hide'} 
  timeAsSystemTime : Tc2_Utilities.TIMESTRUCT; // Actual time as timestring
	{attribute 'hide'} 
	timeAsString : STRING; // Actual time as string
	{attribute 'hide'} 
	LogCache : DynamicStringBuffer; // Dynamic string buffer to cache logs to be processed
	{attribute 'hide'} 
	startLoggingConfiguration : BOOL; // Aux variable to provide fluent interface.
	{attribute 'hide'} 
	internalErrorOccured : BOOL; // Aux variable to log internal errors to Error-property.
	{attribute 'hide'}                                                        				
	_config : ST_LoggingConfiguration; // Logging configuration. Is set by invoking configuration methods.
	{attribute 'hide'} 
	_error : ST_Error; // Contains information about internal error.
	{attribute 'hide'} 
	_busy : BOOL; // Logger is busy, typically with writing logs to the file system.
END_VAR                                                     				
VAR CONSTANT                                                	
	DEFAULT_BUFFER_SIZE : UDINT := 1000; // Default buffer size for FIFO.
END_VAR

// Nothing to be done here. Logger works by invoking its methods.
// "RunLogger" contains all the implementation that has to be processed cyclically.

// Builds logging configuration.
// Required to provide a fluent interface.
// Has to be called at the begin of each method that configures the logger.
{attribute 'hide'}
METHOD PRIVATE BuildLoggingConfiguration : BOOL
IF NOT startLoggingConfiguration THEN
	startLoggingConfiguration := TRUE;
	
	_config.RollingInterval := E_RollingInterval.DAILY;
	_config.WriteToAds := FALSE;
	_config.FileName := '';
	_config.FilePath := 'c:\';
	_config.MinimumLevel := E_LogLevel.DEBUG;
	_config.Delimiter := '|';
	_config.IncludeInstancePath := FALSE;
	_config.LogFileLifespan := 0;
	_config.TimestampFormat := 'YYYYMMDD_hhmm_';
END_IF
END_METHOD

{attribute 'monitoring':='call'}
PROPERTY Busy : BOOL
GET
Busy := _busy;
END_GET
SET // PRIVATE
_busy := Busy;
END_SET
END_PROPERTY

// Returns the current configuration of the logger.
{attribute 'monitoring':='call'}
PROPERTY Configuration : ST_LoggingConfiguration
GET
Configuration := _config;
END_GET
END_PROPERTY

// Configuration method.
// Sets the lifespan of log files. Once exceeded, they will be deleted.
METHOD DeleteLogFilesAfterDays : REFERENCE TO TcLogCore
VAR_INPUT
	Lifespan : UINT; // Lifespan of logfiles in days. Once exceeded, log files will be deleted.
END_VAR
BuildLoggingConfiguration();

_config.LogFileLifespan := Lifespan;

DeleteLogFilesAfterDays REF= THIS^;
END_METHOD

// Returns information about internal errors.
{attribute 'monitoring':='call'}
PROPERTY Error : REFERENCE TO ST_Error
GET
Error REF= _error;
END_GET
END_PROPERTY

{attribute 'hide'} 
METHOD FB_init : BOOL
VAR_INPUT
	bInitRetains : BOOL; // if TRUE, the retain variables are initialized (warm start / cold start)
	bInCopyCode : BOOL;  // if TRUE, the instance afterwards gets moved into the copy code (online change)
	nBufferSize : DINT;  // Buffer size for string buffer
END_VAR
LoggingSingleton.Init(THIS^);
LogCache.Init(DINT_TO_UDINT(nBufferSize));
END_METHOD

{attribute 'hide'} 
METHOD FB_reinit : BOOL
VAR_INPUT
	nBufferSize : DINT; // Buffer size for string buffer
END_VAR
LoggingSingleton.Init(THIS^);
LogCache.Init(DINT_TO_UDINT(nBufferSize));
END_METHOD

METHOD FlushCache : BOOL
LogCache.FlushCache();
END_METHOD

// Configuration method.
// Specifies, if instance path should be included in log file.
METHOD IncludeInstancePath : REFERENCE TO TcLogCore
BuildLoggingConfiguration();

_config.IncludeInstancePath := TRUE;

IncludeInstancePath REF= This^;
END_METHOD

// Logger method.
// Logs data in custom format. No additional formatting will be done.
METHOD LogCustomFormat : BOOL
VAR_INPUT
	Data : Tc2_System.T_MaxString; // Data to be logged. No additional formatting will be done.
END_VAR
IF _config.WriteToAds THEN 
	ADSLOGSTR(ADSLOG_MSGTYPE_LOG OR ADSLOG_MSGTYPE_HINT, Data, ''); 
END_IF

IF _config.FileName <> '' THEN 
	LogCache.AddLine(Data);
END_IF
END_METHOD

// Logger method.
// Logs in the standard format. This includes
// - timestamp
// - log level
// - log message
// - instance path of logging source (optional)
// The message will only be logged if the logging level exceeds the configured minimum logging level.
METHOD LogStandardFormat : BOOL
VAR_INPUT
	Data : Tc2_System.T_MaxString; // Data to be logged. Additional formatting wil be done.
	InstancePath : Tc2_System.T_MaxString; // Instance path of calling logger to locate source of logging message.
	LogLevel : E_LogLevel; // Log level of message.
END_VAR
VAR_INST
	_StringBuilder : StringBuilder;
END_VAR
IF LogLevel >= _config.MinimumLevel THEN
	IF _config.WriteToAds THEN 
		ADSLOGSTR(
			ADSLOG_MSGTYPE_LOG OR LogLevel_To_AdsLogMsgType(LogLevel), 
			_StringBuilder
				.Reset()
				.AppendIf(_config.IncludeInstancePath, InstancePath)
				.AppendIf(_config.IncludeInstancePath, _config.Delimiter)
				.Append(Data)
				.ToString(), 
			''
		); 
	END_IF
	
	IF _config.FileName <> '' THEN 
		LogCache.AddLine(
			_StringBuilder
					.Reset()
					.Append(timeAsString)
					.Append(_config.Delimiter)
					.Append(TO_STRING(LogLevel))
					.AppendIf(_config.IncludeInstancePath, _config.Delimiter)
					.AppendIf(_config.IncludeInstancePath, InstancePath)
					.Append(_config.Delimiter)
					.Append(Data)
					.ToString()
		);
	END_IF
END_IF
END_METHOD

// Configuration method.
// Sets the minimum log level. Log messages below this level 
// will not be logged.
METHOD MinimumLevel : REFERENCE TO TcLogCore
VAR_INPUT 
	Level : E_LogLevel; // Minimum log level to be logged.
END_VAR
BuildLoggingConfiguration();

_config.MinimumLevel := Level;

MinimumLevel REF=THIS^;
END_METHOD

// Checks the specified rolling interval for the file name.
// Generates new file name if rolling intervall exceeded.
{attribute 'hide'}
METHOD PRIVATE RollingIntervalReached : BOOL
VAR_INPUT
	actualTime : Tc2_Utilities.TIMESTRUCT;
	rollingInterval : E_RollingInterval;
END_VAR
VAR_INST	
	rTrigNewHour : Tc2_Standard.R_TRIG;
	rTrigNewDay : R_TRIG;
	rTrigNewMonth : R_TRIG;
	
	newHour : BOOL;
	newDay 	: BOOL;
	newMonth: BOOL;	
END_VAR
rTrigNewHour(CLK := (actualTime.wMinute = 0 AND actualTime.wSecond = 0), 
	Q => newHour);
rTrigNewDay(CLK := (newHour AND actualTime.wHour = 0), 
	Q => newDay);
rTrigNewMonth(CLK := (newDay AND actualTime.wDay = 1), 
	Q => newMonth);

RollingIntervalReached := 	(newHour 	AND rollingInterval = E_RollingInterval.Hourly) OR
							(newDay 	AND rollingInterval = E_RollingInterval.Daily) 	OR
							(newMonth 	AND rollingInterval = E_RollingInterval.Monthly);
END_METHOD

// Cyclic method of Logger.
// This method has to be executed in every plc cycle and runs 
// all internal methods that have to be executed cyclically.
METHOD RunLogger : BOOL
VAR_INST
	rTrigNewDay : Tc2_Standard.R_TRIG;
	TimeData : GenerateTimeData;
	DeleteExpiredLogFiles : DeleteOldFiles;
	_StringBuilder : StringBuilder;
	timeStamp : STRING; // Timestamp used for filename
END_VAR
// Generate time data (shared state)
TimeData(
	timeAsFileTime 		=> timeAsFileTime,
	timeAsSystemTime 	=> timeAsSystemTime,
	timeAsString		=> timeAsString
	);

// Generate new timestamp for filename
IF RollingIntervalReached(timeAsSystemTime, _config.RollingInterval) OR TimeData.Done THEN
	timeStamp := TimeData.ToString(_config.TimestampFormat);
END_IF

// Delete expired log files
rTrigNewDay(CLK := timeAsSystemTime.wHour = 0);
DeleteExpiredLogFiles(
	StartScan 			:= 	rTrigNewDay.Q AND (_config.LogFileLifespan > 0),
	ExpirationInDays 	:=	_config.LogFileLifespan,
	FilePath			:=	_config.FilePath,
	FileName 			:=	_config.FileName,
	ActualTime 			:= 	utcTimeAsFileTime	
	);
IF DeleteExpiredLogFiles.Error.Active THEN
	internalErrorOccured := TRUE;
	_error := DeleteExpiredLogFiles.Error;
END_IF
		
// Persist logging messages to file
LogCache.PersistToFile(
	_StringBuilder
		.Reset()
		.Append(_config.FilePath)
		.AppendIf(RIGHT(_config.FilePath, 1) <> '\', '\')
		.Append(timeStamp)
		.Append(_config.FileName)
		.ToString()
);
IF LogCache.Error.Active THEN
	internalErrorOccured := TRUE;
	_error := LogCache.Error;
END_IF

// Forward busy state of LogCache 
Busy := LogCache.Busy;

// Reset Logging configuration: neccesary in order to provide fluent interface
startLoggingConfiguration := FALSE;

// Reset error flag each cycle to automatically confirm errors once they are gone.
IF NOT internalErrorOccured THEN
	_error.Active := FALSE;
	_error.Code := E_ErrorCode.None;
	_error.Info := '';
END_IF
internalErrorOccured := FALSE;
END_METHOD

// Configuration method
// Sets delimiter between different columns of log file.
METHOD SetDelimiter : REFERENCE TO TcLogCore
VAR_INPUT
	Delimiter : STRING(1); // Delimiter between different columns of log file.
END_VAR
BuildLoggingConfiguration();

_config.Delimiter := Delimiter;

SetDelimiter REF=THIS^;
END_METHOD

// Configuration method
// Sets the rolling interval of the log file. Once the rolling interval
// expires, a file name with a new timestamp will be generated.
METHOD SetRollingInterval : REFERENCE TO TcLogCore
VAR_INPUT
	Interval : E_RollingInterval;	// Rolling interval for log file. Once exceeded, a new log file will be created.
END_VAR
BuildLoggingConfiguration();

_config.RollingInterval := Interval;

SetRollingInterval REF= THIS^;
END_METHOD

// Configuration method
// Sets the format of the timestamp in the file name.
METHOD TimestampFormat : REFERENCE TO TcLogCore
VAR_INPUT
	Format : STRING; // Format the timestamp should have
END_VAR
BuildLoggingConfiguration();

_config.TimestampFormat := Format;

TimestampFormat REF= THIS^;
END_METHOD

// Configuration method.
// Writes logdata to ADS log.
METHOD WriteToAds : REFERENCE TO TcLogCore
BuildLoggingConfiguration();

_config.WriteToAds := TRUE;

WriteToAds REF= This^;
END_METHOD

// Configuration method.
// Writes log message to file.
METHOD WriteToFile : REFERENCE TO TcLogCore
VAR_INPUT
	Path : Tc2_System.T_MaxString; // File path to be written to. Has to end with '\'.
	FileName : STRING; // File name to be written to. Will automatically be prefixed by timestamp.
END_VAR
BuildLoggingConfiguration();

_config.FilePath := Path;
_config.FileName := FileName;

WriteToFile REF= This^;
END_METHOD

END_FUNCTION_BLOCK

// ---- StringBuilder/StringBuilder.TcPOU
FUNCTION_BLOCK PUBLIC StringBuilder IMPLEMENTS IStringBuilder, ILimitedStringBuilder
VAR
	{attribute 'hide'}
	_workString : Tc2_System.T_MaxString;
END_VAR

// Source:

METHOD PUBLIC Append : IStringBuilder // Append text to t current build string.
VAR_INPUT
	text : Tc2_System.T_MaxString; //Text to append to current build string
END_VAR
_workString:= Concat(_workString,text);
Append := THIS^;
END_METHOD

METHOD PUBLIC AppendIf : IStringBuilder
VAR_INPUT
	condition	:	BOOL;
	text : Tc2_System.T_MaxString;
END_VAR
IF condition THEN
	_workString:= Concat(_workString,text);
END_IF
AppendIf := THIS^;
END_METHOD

METHOD PUBLIC InsertAtLocation : IStringBuilder
VAR_INPUT
	Text : Tc2_System.T_MaxString;
	Position:INT;
END_VAR
_workString := Tc2_Standard.INSERT(_WorkSTring,Text,Position);
InsertAtLocation  := THIS^;
END_METHOD

METHOD PadLeft : IStringBuilder
VAR_INPUT
	text : Tc2_System.T_MaxString; // Text to append to current build string
	length : INT; // Total length of text + padding
	char : STRING(1);	// Character to be padded left of text
END_VAR
VAR
	i	: INT;
	padLength : INT;
END_VAR
// Add left padding
padLength := LEN(text) - length;
FOR i := 1 TO padLength DO
	_workString:= Concat(_workString, char);
END_FOR

// Add text
_workString:= Concat(_workString,text);

PadLeft := THIS^;
END_METHOD

METHOD PUBLIC Reset : ILimitedStringBuilder //Reset current build string to an empty string.
_workString:='';
Reset := THIS^;
END_METHOD

METHOD PUBLIC ToString : Tc2_System.T_MaxString //Returns current build string.
ToString := _workString;
END_METHOD

END_FUNCTION_BLOCK

// ---- Logger/POU/TcLogTRIG.TcPOU
FUNCTION_BLOCK TcLogTRIG EXTENDS TcLog

// Logs data on falling edge of CLK.
METHOD OnFallingEdge : REFERENCE TO TcLog
VAR_INPUT
	CLK : BOOL;	// Falling edge logs data.
END_VAR
VAR_INST
	fTrig	:	Tc2_Standard.F_TRIG;
END_VAR
fTrig(CLK:=CLK);

SUPER^.OnCondition(fTrig.Q);

OnFallingEdge REF= THIS^;
END_METHOD

// Logs data on rising edge of CLK.
METHOD OnRisingEdge : REFERENCE TO TcLog
VAR_INPUT
	CLK : BOOL; // Rising edge logs data.
END_VAR
VAR_INST
	rTrig	:	Tc2_Standard.R_TRIG;
END_VAR
rTrig(CLK:=CLK);

SUPER^.OnCondition(rTrig.Q);

OnRisingEdge REF= THIS^;
END_METHOD

END_FUNCTION_BLOCK
